Staubli VAL3: onF4Event.pgx

program onF4Event(bool& x_bSave[])
  local num l_nSize
  local num i
  local TrajectoryItem l_tTraj
  local num l_nTemp
begin
  // look if the bButton is enable
  if bButton[3]
    //
    // paste
    //
    call trajType:getSizeItem(false,l_nSize)
    l_nTemp=nIndex+1
    for i=0 to (l_nSize-1)
      call trajType:getTrajItem(l_tTraj,i)
      if find(l_tTraj.comment,"#")!=-1
        // insert user value
        call trajType:insertItem(i,l_nTemp)
        if i==-1
          return
        else
          // overWrite
          l_tTraj.comment=right(l_tTraj.comment,len(l_tTraj.comment)-1)
          call trajType:setTrajItem(l_tTraj,l_nTemp)
          if l_nTemp<=i
            i=i+1
          endIf
          l_nTemp=l_nTemp+1
          l_nSize=l_nSize+1
        endIf
      endIf
    endFor
    // unselect ALL
    call unSelectItem()
    x_bSave=true
  endIf
end
